FUNCTION_BLOCK TcA2B2Kitten
VAR_INPUT
END_VAR
VAR_OUTPUT
END_VAR
VAR
	_httpClient:			FB_IotHttpClient;
	_httpRequest:			FB_IotHttpRequest;
	_httpRequestHeader:		FB_IotHttpHeaderFieldMap;
	bSendGet:				BOOL;
	connectNow: 			BOOL;
	requestNow: 			BOOL;
	sContent				: STRING(2000);
	configClientConnect: BOOL;
	getContentNow: BOOL;
	
	_jsonDomParser : FB_JsonDomParser;
	jsonRoot : SJsonValue;
	jsonProp : SJsonValue;
	parseContentNow: BOOL;
	sState: STRING;
	
	
	_jsonSaxParser : 				FB_JsonSaxReader;
	jsonSaxHandler_RobotState :		JsonSaxHandler_RobotState;
	
	saxParseContentNow: 			BOOL;
END_VAR


IF configClientConnect THEN 
	//_httpClient.sHostName := '192.168.56.1';
	_httpClient.sHostName := '127.0.0.1';
	_httpClient.nHostPort := 80;
	_httpClient.bKeepAlive := TRUE;
	_httpClient.stTLS.bNoServerCertCheck:=TRUE;
	_httpClient.tConnectionTimeout := T#10S;
	
	configClientConnect := FALSE;
END_IF

IF connectNow THEN
	_httpClient.Execute();
END_IF



//IF _httpClient.bConnected AND requestNow THEN
IF requestNow THEN
	//_httpRequest.eCompressionMode := ;
	//_httpRequest.sContentType := ;
	
	_httpRequestHeader.AddField('accept', 'application/hal+json;v=2.0', FALSE);
	_httpRequestHeader.AddField('authorization', 'Basic RGVmYXVsdCBVc2VyOnJvYm90aWNz', FALSE);	// encoded Username: Default User, Password: robotics
	
	_httpRequest.SendRequest(sUri:='/rw/rapid/execution', fbClient:=_httpClient, eRequestType:=ETcIotHttpRequestType.HTTP_Get, pContent:=0, nContentSize:=0, fbHeader:=_httpRequestHeader);
	
	requestNow := FALSE;
END_IF


IF getContentNow THEN
	_httpRequest.GetContent(ADR(sContent), nContentSize:=SIZEOF(sContent), TRUE);
	getContentNow := FALSE;
END_IF


IF parseContentNow THEN
	jsonRoot := _jsonDomParser.ParseDocument(sContent);
	jsonProp := _jsonDomParser.FindMemberPath(jsonRoot, 'state#0/ctrlexecstate');	// See https://infosys.beckhoff.com/english.php?content=../content/1033/tcplclib_tc3_jsonxml/3664369803.html&id=4049129407046606983
	IF (jsonProp <> 0) THEN
  		sState := _jsonDomParser.GetString(jsonProp);
	END_IF
	
	parseContentNow := FALSE; 
END_IF


IF saxParseContentNow THEN
	jsonSaxHandler_RobotState.Reset();
	_jsonSaxParser.Parse(sContent, ipHdl := jsonSaxHandler_RobotState, );
	sState := jsonSaxHandler_RobotState.parsedState;
	
	saxParseContentNow := FALSE; 
END_IF

END_FUNCTION_BLOCK

(* stored: Version 1.1.0.1, ProductVersion 3.1.4024.12
   POU TcA2B2Kitten: Id {ea1fde4a-6390-43d8-ae6c-e82c42f674c2}, SpecialFunc None *)
